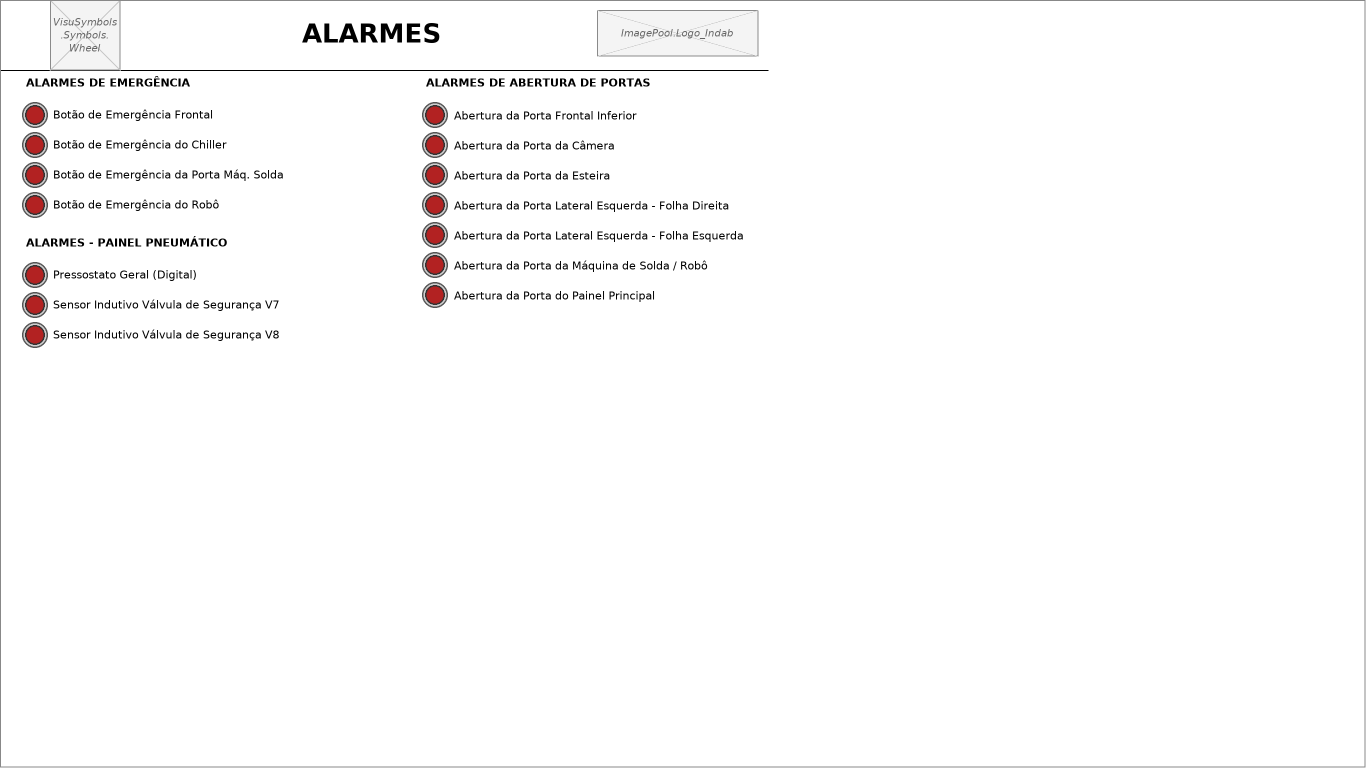
VISUALIZATION Tela_Alarmes_1  // 1366x768
    Line (0,70) (768,70)
    Line (0,1312) (768,1312)
    Image (597,10 161x46), image: ImagePool.Logo_Indab
    Rectangle (584,1340 180x24), "%t[dd/MM/yyyy]"
    Rectangle (584,1316 180x24), "%t[HH:mm:ss]"
    Label (153,7 437x53), "ALARMES"
    Lamp1 (20,100 30x30), variable: Alarmes.ByteAlarmeEmergencia.0, style: Lamp-Lamp1-Red
    Rectangle (50,100 250x30), "Botão de Emergência Frontal"
    Lamp1 (20,130 30x30), variable: Alarmes.ByteAlarmeEmergencia.1, style: Lamp-Lamp1-Red
    Rectangle (50,130 250x30), "Botão de Emergência do Chiller"
    Lamp1 (20,160 30x30), variable: Alarmes.ByteAlarmeEmergencia.2, style: Lamp-Lamp1-Red
    Rectangle (50,160 250x30), "Botão de Emergência da Porta Máq. Solda"
    Lamp1 (20,190 30x30), variable: Alarmes.ByteAlarmeEmergencia.3, style: Lamp-Lamp1-Red
    Rectangle (50,190 250x30), "Botão de Emergência do Robô"
    Rectangle (23,73 237x20), "ALARMES DE EMERGÊNCIA"
    Lamp1 (420,100 30x30), variable: Alarmes.ByteAlarmeAberturaPortas.0, style: Lamp-Lamp1-Red
    Rectangle (451,101 300x30), "Abertura da Porta Frontal Inferior"
    Lamp1 (420,130 30x30), variable: Alarmes.ByteAlarmeAberturaPortas.1, style: Lamp-Lamp1-Red
    Rectangle (451,131 300x30), "Abertura da Porta da Câmera"
    Lamp1 (420,160 30x30), variable: Alarmes.ByteAlarmeAberturaPortas.2, style: Lamp-Lamp1-Red
    Rectangle (451,161 300x30), "Abertura da Porta da Esteira"
    Lamp1 (420,190 30x30), variable: Alarmes.ByteAlarmeAberturaPortas.3, style: Lamp-Lamp1-Red
    Rectangle (451,191 300x30), "Abertura da Porta Lateral Esquerda - Folha Direita"
    Lamp1 (420,220 30x30), variable: Alarmes.ByteAlarmeAberturaPortas.4, style: Lamp-Lamp1-Red
    Rectangle (451,221 300x30), "Abertura da Porta Lateral Esquerda - Folha Esquerda"
    Lamp1 (420,250 30x30), variable: Alarmes.ByteAlarmeAberturaPortas.5, style: Lamp-Lamp1-Red
    Rectangle (451,251 300x30), "Abertura da Porta da Máquina de Solda / Robô"
    Lamp1 (420,280 30x30), variable: Alarmes.ByteAlarmeAberturaPortas.6, style: Lamp-Lamp1-Red
    Rectangle (451,281 300x30), "Abertura da Porta do Painel Principal"
    Rectangle (423,73 237x20), "ALARMES DE ABERTURA DE PORTAS"
    Button (15,1315 175x45), "RECEITAS"
        OnMouseClick: change screen: Tela_Receita
    Lamp1 (20,260 30x30), variable: Alarmes.ByteAlarmePainelPneumatico.0, style: Lamp-Lamp1-Red
    Rectangle (50,260 250x30), "Pressostato Geral (Digital)"
    Lamp1 (20,290 30x30), variable: Alarmes.ByteAlarmePainelPneumatico.1, style: Lamp-Lamp1-Red
    Rectangle (50,290 250x30), "Sensor Indutivo Válvula de Segurança V7"
    Lamp1 (20,320 30x30), variable: Alarmes.ByteAlarmePainelPneumatico.2, style: Lamp-Lamp1-Red
    Rectangle (50,320 250x30), "Sensor Indutivo Válvula de Segurança V8"
    Rectangle (23,233 237x20), "ALARMES - PAINEL PNEUMÁTICO"
    Image (50,0 70x70), image: VisuSymbols.Symbols.Wheel
        OnMouseClick: change screen: Tela_Alarmes_2
    Button (375,1315 175x45), "PRODUÇÃO"
        OnMouseClick: change screen: Tela_Producao
    Button (195,1315 175x45), "MANUTENÇÃO"
        OnMouseClick: change screen: Tela_Manutencao
END_VISUALIZATION

(* stored: Version 1.1.0.1, ProductVersion 3.1.4024.11
   Visu Tela_Alarmes_1: Id {95bc2723-c044-4c36-82a5-95b0dd9529ee} *)
